// TIA Portal V17 export
// export: Created 2023-02-13T11:16:36.1295977Z, ExportSetting WithDefaults, DisplayName Totally Integrated Automation Portal, DisplayVersion V17, DisplayName TIA Portal Openness, DisplayVersion V17, DisplayName TIA Portal Teamcenter Gateway, DisplayVersion V17, DisplayName TIA Portal Version Control Interface, DisplayVersion V17, DisplayName SINAMICS Startdrive Advanced, DisplayVersion V17, DisplayName SINAMICS Startdrive G130, G150, S120, S150, SINAMICS MV, S210, DisplayVersion V17, DisplayName SINAMICS Startdrive G110M, G120, G120C, G120D, G120P, G115D, DisplayVersion V17, DisplayName STEP 7 Professional, DisplayVersion V17, DisplayName STEP 7 Safety, DisplayVersion V17, DisplayName WinCC Professional, DisplayVersion V17
DATA_BLOCK "Totalizer_FT-03.01"   // DB383
VERSION : 0.1
// stored: AutoNumber false, DBAccessibleFromOPCUA true, DBAccessibleFromWebserver true, InstanceOfName Totalizer, InstanceOfType FB
"Totalizer"
   // VAR_INPUT
   //    value : Real;
   //    intervall : Time;
   //    cycle : Time;
   //    reset : Bool;
   // END_VAR
   // VAR_OUTPUT
   //    total : Real;
   // END_VAR
   // VAR
   //    statAccum : Real;
   // END_VAR
BEGIN
END_DATA_BLOCK
